TYPE Buffer_Cnv_Settings_DUT :
STRUCT
	ID:	DINT;
	Barcode_ID:	UINT;
	Cnv_Level:	UINT;
	TC_Time:	UINT;
	Transfer_Time:	UINT;
	Pallet_Align_Time:	UINT;
	Slow_Speed:	UINT;
	Full_Speed:	UINT;
	Manual_Speed:	UINT;
	Safety_stop_Timeout:	UINT;
END_STRUCT
END_TYPE

(* stored: Version 1.1.0.1
   DUT Buffer_Cnv_Settings_DUT: Id {a189004e-295e-4110-a348-44d8e744c89c} *)
